{attribute 'qualified_only'}
{attribute 'strict'}
TYPE E_MainState :
(
	RUN		:=	0,
	STOP	:=	1,
	PAUSE	:=	2,
	FAULT	:=	3
);
END_TYPE

(* stored: Version 1.1.0.1, ProductVersion 3.1.4024.16
   DUT E_MainState: Id {9299ab1f-b2d8-47b7-813c-a32b914e675d} *)
